// TIA Portal V16 export
// export: Created 2021-07-12T14:47:20.7741622Z, ExportSetting WithDefaults, DisplayName Totally Integrated Automation Portal, DisplayVersion V16, DisplayName TIA Portal Version Control Interface, DisplayVersion V16, DisplayName TIA Portal Openness, DisplayVersion V16, DisplayName STEP 7 Professional, DisplayVersion V16, DisplayName STEP 7 Safety, DisplayVersion V16, DisplayName WinCC Professional, DisplayVersion V16
TYPE "SimaHydTO_typeHMIConnectionVCharEditor"
TITLE = SimaHydTO_typeHMIConnectionVCharEditor
// HMI interface: VChar editor
// stored: IsFailsafeCompliant false
   STRUCT
      Command { S7_SetPoint := 'True'} : "SimaHydTO_typeHMIConnectionVCharEditorCommand";   // Data: HMI -> PLC
      Status { S7_SetPoint := 'True'} : "SimaHydTO_typeHMIConnectionVCharEditorStatus";   // Data: PLC -> HMI
      Parameter { S7_SetPoint := 'True'} : "SimaHydTO_typeHMIConnectionVCharEditorParameter";   // Data: PLC <-> HMI (Load and save)
      Table { S7_SetPoint := 'True'} : "SimaHydTO_typeHMIConnectionVCharEditorTable";   // Data table of VChar
      VCharNameToSave : WString[24];   // Name of VChar to be saved
   END_STRUCT;
END_TYPE
